                                                    IF Globals.enableDryCycle THEN
                                                        Globals.dryCycleCount := Globals.dryCycleCount + 1;     
                                                    ELSE
                                                        Globals.bagsMadeCount := Globals.bagsMadeCount + 1; 
                                                    END_IF
													IF enableBagOpen THEN
                                                        state := HEAD_STATES.OpenBag;
                                                    ELSE
                                                        state := HEAD_STATES.FinishCycle;
                                                    END_IF
                                                    
                                                            
                                                    
                                
    HEAD_STATES.OpenBag :                            // Close jaw to grab the bag
                                                    openBagSubState := BAG_OPEN_ASSIST_STATES.MoveJawIn;
                                                    state := HEAD_STATES.OpeningBag;
                                                    
                                                    
    HEAD_STATES.OpeningBag :                        // Open jaw and grab onto the bag
                                                    IF openBagSubState = BAG_OPEN_ASSIST_STATES.Done THEN
                                                        state := HEAD_STATES.OpenedBag;
                                                        openBagSubState := BAG_OPEN_ASSIST_STATES.Idle;
													ELSIF openBagSubState = BAG_OPEN_ASSIST_STATES.FeedNewBag THEN
														state := HEAD_STATES.SealAndSeparateBag;
														openBagSubState := BAG_OPEN_ASSIST_STATES.Idle;
                                                    END_IF
                                                    
    HEAD_STATES.OpenedBag :                            // Move fingers in and to bag holding and reset cycle
                                                    IF (motorizedSealFlatteners.state = SEAL_FLATTENER_STATES.Idle OR NOT motorizedSealFlatteners.enable) //OR bagFailedToOpen
														 AND pressureBar.state = PRESSURE_BAR_STATES.JawOpened THEN
														state := HEAD_STATES.FinishCycle;
                                                    END_IF
	HEAD_STATES.FinishCycle :			//
													finishCycleSubState := FINISH_CYCLE_STATES.Start;
													state := HEAD_STATES.FinishingCycle;
	HEAD_STATES.FinishingCycle : 		//
													IF finishCycleSubState = FINISH_CYCLE_STATES.Done THEN
														state := HEAD_STATES.FinishedCycle;
														finishCycleSubState := FINISH_CYCLE_STATES.Idle;
													END_IF
	HEAD_STATES.FinishedCycle :			//
											HMIData.bagsMade.Increment();
											HMIData.resettableBagsMade.Increment();
                                            state := HEAD_STATES.Idle;
											filler.BaggerCycledAndReady();
											cycleTime := (TIME_TO_REAL(cycleTimer.ET) / 1000); 
											cycleTimer.IN := FALSE;
											IF HMIData.averageCycleTime = 0 THEN
												HMIData.averageCycleTime := cycleTime;
											ELSE
												HMIData.averageCycleTime := (cycleTime + HMIData.averageCycleTime) / 2;
											END_IF
											HMIData.inCycle := FALSE;
											//bagFailedToOpen := FALSE;
											IF HMIData.factoryTestMode AND NOT HMIData.stopMachine THEN
												IF (HMIData.bagsMade.count >= 1000) THEN
													factoryTestModeKeepCycling := FALSE;
													HMIData.factoryTestMode := FALSE;
												ELSE
													factoryTestModeKeepCycling := TRUE;
												END_IF
											END_IF	
											
    HEAD_STATES.StartHoming :            // 
                                            passthrough.HomeEndStop();
                                            state := HEAD_STATES.Homing;                                        
    
    HEAD_STATES.Homing :                // 
                                            IF passthrough.state = PASSTHROUGH_SERVO_STATES.HomeComplete THEN
                                                state := HEAD_STATES.HomingComplete;       
                                            END_IF
                                            
    HEAD_STATES.HomingComplete :        // 
                                            homeJawPB := FALSE;
                                            state := HEAD_STATES.Idle;
											//HMIData.passthroughSetting := 6.0;
											setPassthroughPB := TRUE;
    
    HEAD_STATES.MovePassthrough :        // 
                                            pressureBar.AutoMovingPassthrough();
                                            passthrough.MovePassthrough(passthroughSetting);
                                            state := HEAD_STATES.MovingPassthrough;
    
    HEAD_STATES.MovingPassthrough :    IF passthrough.state = PASSTHROUGH_SERVO_STATES.PassthroughMovedIn OR passthrough.state = PASSTHROUGH_SERVO_STATES.PassthroughMovedOut THEN
                                                state := HEAD_STATES.MovedPassthrough;     
                                            END_IF
                                            
    HEAD_STATES.MovedPassthrough :        // 
                                            pressureBar.AutoDoneMovingPassthrough();
                                            state := HEAD_STATES.Idle;
											setPassthroughPB := FALSE;
                                                    
    HEAD_STATES.Fault :                     hmiLight.TurnOff();
											HMIData.inCycle := FALSE;
											cycleTimer.IN := FALSE;
											bagDelivery.bagFeedMasterMotor.SetRearMotorToEncoderFollowing();
											sealAndSeparateSubState := SEAL_SEPARATE_STATES.Idle;
											releaseAndFeedSubState := RELEASE_FEED_STATES.Idle;
											openBagSubState := BAG_OPEN_ASSIST_STATES.Idle;
											finishCycleSubState := FINISH_CYCLE_STATES.Idle;
											oVacOn := FALSE;
											filler.Reset();
											LPA.ManualOff();
											IBDRetractToDeflate.Reset();
											IBDRetractToEject.Reset();
											exitConveyorRun.Reset();
											externalExitConveyorRun.Reset();
											oRunPrinterRibbonUnwindMotor := FALSE;
											setPassthroughPB := FALSE;
											homeJawPB := FALSE;
											startCycle := FALSE;
											HMIData.initiateCycle := FALSE;
											factoryTestModeKeepCycling := FALSE;
											pressureBarCloseDelay.IN := FALSE;
											//bagOpened := FALSE;
                                                    
END_CASE

CASE sealAndSeparateSubState OF
    SEAL_SEPARATE_STATES.Idle : 
	
	SEAL_SEPARATE_STATES.BringInIBD : 				// Bring in IBD if enabled
													IF enableIBDDeflate THEN
														IBDRetractToDeflate.Trigger();
													END_IF 
													
													sealAndSeparateSubState := SEAL_SEPARATE_STATES.WaitForJawCloseDelay;
	
	SEAL_SEPARATE_STATES.WaitForJawCloseDelay : 	// Wait for jaw close delay. 
													IF pressureBar.enable THEN
														LPA.ManualOff();
														pressureBarCloseDelay.IN := TRUE;
														IF (pressureBarCloseDelay.Q OR HMIData.pressureBarCloseDelay = 0)
															AND (funnel.closed OR NOT funnel.enable)
															THEN
															sealAndSeparateSubState := SEAL_SEPARATE_STATES.MoveJawIn;
															pressureBarCloseDelay.IN := FALSE;
														END_IF
                                                    ELSE 
                                                        sealAndSeparateSubState := SEAL_SEPARATE_STATES.ReverseBag;
                                                    END_IF
        
    SEAL_SEPARATE_STATES.MoveJawIn :                // Perform actions as enabled - close jaw and move flatteners out. If jaw is disabled then go right to reverse bag
                                                    IF motorizedSealFlatteners.enable THEN
                                                        motorizedSealFlatteners.AutoMoveOut();
                                                    END_IF
                                                    
													pressureBar.AutoCloseJaw();
                                                    sealAndSeparateSubState := SEAL_SEPARATE_STATES.MovingJawIn;
                                                    
                                                    
                                                    
                                                    
                                                    
    SEAL_SEPARATE_STATES.MovingJawIn :                // If Jaw is in and flatteners out then move on
                                                    IF (motorizedSealFlatteners.state = SEAL_FLATTENER_STATES.MovedFlattenersOut OR NOT motorizedSealFlatteners.enable) 
                                                        AND (pressureBar.state = PRESSURE_BAR_STATES.JawClosed OR NOT pressureBar.enable)
                                                        THEN
                                                            sealAndSeparateSubState := SEAL_SEPARATE_STATES.MovedJawIn;    
                                                    END_IF
                                                                
    SEAL_SEPARATE_STATES.MovedJawIn :                // Will add sealing logic here
                                                    sealAndSeparateSubState := SEAL_SEPARATE_STATES.ReverseBag;
                                                    
    SEAL_SEPARATE_STATES.ReverseBag :                // Reverse bag if bag delivery enabled, otherwise open jaw
													IBDRetractToDeflate.Reset();
                                                    IF bagDelivery.enable THEN
                                                        bagDelivery.AutoReverseBag();
                                                        sealAndSeparateSubState := SEAL_SEPARATE_STATES.ReversingBag;
                                                    ELSE sealAndSeparateSubState := SEAL_SEPARATE_STATES.Done;    
                                                    END_IF
                                                                    
    SEAL_SEPARATE_STATES.ReversingBag :                // 
													IF NOT HMIData.separateBeforeSeal THEN
														sealTimer.PT := TO_TIME(HMIData.sealBarDwell * 1000);
														sealTimer.IN := TRUE;
														IF NOT sealTimer.Q THEN
															oSealBarExtend := TRUE;
															oSealBarRetract := FALSE;
														ELSE 
															
															oSealBarExtend := FALSE;
															oSealBarRetract := TRUE;
															
														END_IF
													END_IF

                                                    IF (motorizedSealFlatteners.state = SEAL_FLATTENER_STATES.MovedFlattenersOut OR NOT motorizedSealFlatteners.enable) 
                                                        AND (pressureBar.state = PRESSURE_BAR_STATES.JawClosed OR NOT pressureBar.enable)
                                                        AND (bagDelivery.state = BAG_DELIVERY_STATES.ReverseDone OR NOT bagDelivery.enable)
														AND (sealTimer.Q OR HMIData.separateBeforeSeal)
                                                        THEN
															IF NOT HMIData.separateBeforeSeal THEN
																HMIData.sealBarCycles.Increment();
															END_IF
															
															sealTimer.IN := FALSE;
                                                            sealAndSeparateSubState := SEAL_SEPARATE_STATES.Reversedbag;
                                                    END_IF
    SEAL_SEPARATE_STATES.Reversedbag :                // 
                                                    sealAndSeparateSubState := SEAL_SEPARATE_STATES.SealBag;
													
	SEAL_SEPARATE_STATES.SealBag:					
													IF HMIData.separateBeforeSeal THEN
														sealTimer.PT := TO_TIME(HMIData.sealBarDwell * 1000);
														sealTimer.IN := TRUE;
														IF NOT sealTimer.Q THEN
															oSealBarExtend := TRUE;
															oSealBarRetract := FALSE;
														ELSE 
															sealTimer.IN := FALSE;
															oSealBarExtend := FALSE;
															oSealBarRetract := TRUE;
															HMIData.sealBarCycles.Increment();
															sealAndSeparateSubState := SEAL_SEPARATE_STATES.Done;
														END_IF
													ELSE
														sealAndSeparateSubState := SEAL_SEPARATE_STATES.Done;
													END_IF
													
																				
                                                    
    SEAL_SEPARATE_STATES.Done :                        // 
                                                    
                                    
    SEAL_SEPARATE_STATES.Fault :
END_CASE


CASE releaseAndFeedSubState OF
    RELEASE_FEED_STATES.Idle :                        //
                                                        
    RELEASE_FEED_STATES.MoveJawOutAndDropBag :        // 
                                                    IF (motorizedSealFlatteners.state = SEAL_FLATTENER_STATES.MovedFlattenersOut OR NOT motorizedSealFlatteners.enable) 
                                                        AND (pressureBar.state = PRESSURE_BAR_STATES.JawClosed OR NOT pressureBar.enable)
                                                        AND ((bagDelivery.state = BAG_DELIVERY_STATES.ReverseDone) OR Globals.enableDryCycle)
                                                        OR (bagDelivery.state =  BAG_DELIVERY_STATES.WaitingForPrinter AND zebraPrinter.enable)
                                                        OR NOT bagDelivery.enable
                                                        THEN
                                                            IF motorizedSealFlatteners.enable THEN
                                                                motorizedSealFlatteners.AutoMoveToClearance();
                                                            END_IF
                                                            
                                                            IF pressureBar.enable THEN
                                                                pressureBar.AutoOpenJaw();
                                                            END_IF
                                                            
															IF enableBagOpen THEN
																bagOpenFingers.Release();
															END_IF
															
															IF enableIBDEject THEN
																IBDRetractToEject.Trigger();
															END_IF
															
															IF enableLoadPlate THEN
																rearLoadPlateRetract.Trigger();
															END_IF
															
															IF TO_DINT(HMIData.exitConveyorDwell) <> 0 THEN
																exitConveyorRun.Trigger();
															END_IF
															
															IF TO_DINT(HMIData.externalExitConveyorDwell) <> 0 THEN
																externalExitConveyorRun.Trigger();
															END_IF
															
															IF enableLabelSideUp THEN
																forwardLoadPlateRetract.Trigger();
																loadShelfExtend.Trigger();
															END_IF
															
															IF HMIData.lpaBagEjectAssistEnable THEN
																LPA.ManualOn();
															END_IF
                                                           bagDropTimer.IN := TRUE;
														   releaseAndFeedSubState := RELEASE_FEED_STATES.MovingJawOutAndDroppingBag;
                                                    END_IF
													
	 RELEASE_FEED_STATES.MovingJawOutAndDroppingBag :
														 // If printer is enabled then perform printer operation of bag delivery, otherwise just feed new bag out.
                                                            // In the case that bagDelivery is disabled then we're done with release and feed
                                                        IF bagDropTimer.Q 
															AND (motorizedSealFlatteners.state = SEAL_FLATTENER_STATES.MovedFlattenersToBagFeed OR NOT motorizedSealFlatteners.enable)
															THEN   
															bagDropTimer.IN := FALSE;
															IBDRetractToEject.Reset();
															IBDRetractToDeflate.Reset();
															IF bagDelivery.enable AND NOT zebraPrinter.enable THEN
                                                                bagDelivery.AutoFeedBagOut();
																LPA.ManualOff();
																IF HMIData.lpaDuringBagFeedEnable THEN
																	LPA.ManualOn();
																END_IF
                                                                releaseAndFeedSubState := RELEASE_FEED_STATES.MovingJawOutAndFeedingBag;
                                                            ELSIF bagDelivery.enable AND zebraPrinter.enable THEN
                                                                bagDelivery.AutoWaitForPrinter();
																LPA.ManualOff();
                                                                releaseAndFeedSubState := RELEASE_FEED_STATES.WaitForPrinter;
                                                            ELSE 
                                                                releaseAndFeedSubState := RELEASE_FEED_STATES.Done;
                                                            END_IF
                                                            (*{warning 'TODO: This is a hack to use HPA as LPA'}
														    HPA.DwellSetting := 500;		// Get rid on this - ha
													        HPA.Trigger();*)												
    													END_IF
														
    RELEASE_FEED_STATES.WaitForPrinter :            // Data Ready means the printer has a label and we're all set to print
                                                    IF zebraPrinter.state = PRINTER_STATES.DataReady THEN
                                                        releaseAndFeedSubState := RELEASE_FEED_STATES.FeedToOffset;
                                                    END_IF
                                                    
    RELEASE_FEED_STATES.FeedToOffset :                // This starts feeding to the print offset
													IF (motorizedSealFlatteners.state = SEAL_FLATTENER_STATES.MovedFlattenersToBagFeed OR NOT motorizedSealFlatteners.enable) THEN
														bagDelivery.AutoPrinterReady();
                                                    	releaseAndFeedSubState := RELEASE_FEED_STATES.FeedingToOffset;
													END_IF
                                                    
                                                        
    RELEASE_FEED_STATES.FeedingToOffset :            // Once offset done start printing
                                                    IF bagDelivery.state = BAG_DELIVERY_STATES.FedToPrintOffset THEN
                                                        releaseAndFeedSubState := RELEASE_FEED_STATES.StartPrinting;
                                                    END_IF                                            
    
    RELEASE_FEED_STATES.StartPrinting :                // Printer starts print cycle and bag delivery starts moving at print speed
                                                    
                                                    //bagDelivery.AutoStartPrintFeed();
													zebraPrinter.AutoPrintNow();
                                                    
                                                    releaseAndFeedSubState := RELEASE_FEED_STATES.SendPrintSignal;                                            

    RELEASE_FEED_STATES.SendPrintSignal:            // 
                                                    //IF bagDelivery.state =     BAG_DELIVERY_STATES.FeedingAtPrintSpeed THEN
													//zebraPrinter.AutoSendPrintSignal();
													IF zebraPrinter.printHeadDebounced THEN
														bagDelivery.AutoStartPrintFeed();
														zebraPrinter.AutoSendPrintSignal();
														barcodeVerifier.Trigger();
                                                        //bagDelivery.AutoStartPrintFeed();
														//bagDelivery.AutoStartPrintFeed();
                                                        //zebraPrinter.AutoSendPrintSignal();
														
                                                        releaseAndFeedSubState := RELEASE_FEED_STATES.Printing;
                                                    END_IF                                        

    RELEASE_FEED_STATES.Printing :                // 
													
                                                    IF zebraPrinter.state = PRINTER_STATES.DonePrinting THEN
                                                        releaseAndFeedSubState := RELEASE_FEED_STATES.StopPrinting;
                                                    END_IF
                                                    
    RELEASE_FEED_STATES.StopPrinting :                // Tell bag delivery it's okay to feed out the rest of the bag and the printer that it can prep itself for the next print
                                                    bagDelivery.AutoPrinterDone();
                                                    zebraPrinter.AutoAckPrintDone();
													IF HMIData.lpaDuringBagFeedEnable THEN
														LPA.ManualOn();
													END_IF
													
                                                    releaseAndFeedSubState := RELEASE_FEED_STATES.MovingJawOutAndFeedingBag;
                                                                                
                                                                                                            
    RELEASE_FEED_STATES.MovingJawOutAndFeedingBag :    // 
    
													
													IF (bagdelivery.state = BAG_DELIVERY_STATES.Ready OR NOT bagdelivery.enable)
                                                        AND (motorizedSealFlatteners.state = SEAL_FLATTENER_STATES.MovedFlattenersToBagFeed OR NOT motorizedSealFlatteners.enable) 
                                                        AND (pressureBar.state = PRESSURE_BAR_STATES.JawOpened OR NOT pressureBar.enable)
                                                        THEN
															IF LPA.DwellSetting = 0 THEN
																LPA.ManualOff();
															END_IF
															IBDRetractToEject.Reset();
                                                            releaseAndFeedSubState := RELEASE_FEED_STATES.MovedJawOutAndFedBag;
                                                    END_IF
                                                    
    RELEASE_FEED_STATES.MovedJawOutAndFedBag :      // Wait until bag is fed out before triggering barcode fail.
													IF barcodeVerifier.barcodeFault THEN
														barcodeVerificationFailed.Trigger();
													END_IF 
													releaseAndFeedSubState := RELEASE_FEED_STATES.Done;
    RELEASE_FEED_STATES.Done :
    RELEASE_FEED_STATES.Fault :
END_CASE

CASE openBagSubState OF
    BAG_OPEN_ASSIST_STATES.Idle :                    // 
                                                    
                                                    
                                                    
    BAG_OPEN_ASSIST_STATES.MoveJawIn :                // Close jaw against bag. In the future we may also start vacuum here
                                                    pressureBar.AutoCloseJaw();
													(*HPA.DwellSetting := 80;
													HPA.Trigger();*)
													IF HPA.DwellSetting <> 0 THEN
														HPA.Trigger();	
													END_IF
													
													//oVacOn := TRUE; // Hard coded for now, this is vacuum
                                                    openBagSubState := BAG_OPEN_ASSIST_STATES.MovingJawIn;        
                                                    
                                                    
    BAG_OPEN_ASSIST_STATES.MovingJawIn :            // Move on once jaw is closed
                                                    IF (pressureBar.state = PRESSURE_BAR_STATES.JawClosed) OR NOT pressureBar.enable THEN
                                                        openBagSubState := BAG_OPEN_ASSIST_STATES.MovedJawIn;        
                                                    END_IF
                                                    
                                                    
    BAG_OPEN_ASSIST_STATES.MovedJawIn :                // Hold onto the bag with vacuum to build suction
                                                    vacuumHoldTimer.IN := TRUE;
													oVacOn := TRUE; // Hard coded for now, this is vacuum
													IF vacuumHoldTimer.Q THEN
														openBagSubState := BAG_OPEN_ASSIST_STATES.MoveJawOut; 
														vacuumHoldTimer.IN := FALSE;
													END_IF
                                                                   
                                                    
                                                    
    BAG_OPEN_ASSIST_STATES.MoveJawOut :                // Open the jaw and move seal flatteners in and to bag holding
                                                    pressureBar.AutoOpenJaw();
													motorizedSealFlatteners.AutoMoveIn();
                                                    openBagSubState := BAG_OPEN_ASSIST_STATES.MovingJawOutAndGrab;
                                                    
                                                    
    BAG_OPEN_ASSIST_STATES.MovingJawOutAndGrab :    // Once everything that is enabled is homed finish cycle 
													bagOpenFingerDelay.IN := TRUE;
													IF bagOpenFingerDelay.Q THEN
														bagOpenFingers.Grab();
														bagOpenFingerDelay.IN := FALSE;

														openBagSubState := BAG_OPEN_ASSIST_STATES.CheckForSuccessfulBagGrab;
													END_IF
													  

	BAG_OPEN_ASSIST_STATES.CheckForSuccessfulBagGrab : 	//
														IF bagOpenRetryCount < bagOpenRetrySetting THEN
															bagOpenCheckDelay.IN := TRUE;
															IF bagOpenCheckDelay.Q THEN
																IF bagOpenFingers.CheckIfBagGrabbed(TRUE) THEN // This method checks to see if the bag is grabbed and returns true if so.
																	openBagSubState := BAG_OPEN_ASSIST_STATES.BagOpened;
																	motorizedSealFlatteners.AutoMoveIn();
																ELSE 
																	openBagSubState := BAG_OPEN_ASSIST_STATES.BagFailedToOpen;
																END_IF
																bagOpenCheckDelay.IN := FALSE;
															END_IF
														ELSE 
															motorizedSealFlatteners.AutoMoveToBagHolding();
															openBagSubState := BAG_OPEN_ASSIST_STATES.MovingJawOutAfterGrab;
														END_IF
													  
	BAG_OPEN_ASSIST_STATES.BagFailedToOpen :			// 
														bagOpenFingers.Release();
														bagOpenRetryCount := bagOpenRetryCount + 1;
														IF bagOpenRetryCount < bagOpenRetrySetting THEN
															openBagSubState := BAG_OPEN_ASSIST_STATES.MoveJawIn;
														ELSIF HMIData.bagOpenFeedNewBagCount < HMIData.bagOpenFeedNewBagSetting THEN
															HMIData.bagOpenFeedNewBagCount := HMIData.bagOpenFeedNewBagCount + 1;
															bagOpenRetryCount := 0;
															motorizedSealFlatteners.AutoMoveOut();
															oVacOn := FALSE;
															openBagSubState := BAG_OPEN_ASSIST_STATES.FeedNewBag;
															
														ELSE 
															//IF (motorizedSealFlatteners.state = SEAL_FLATTENER_STATES.Idle OR NOT motorizedSealFlatteners.enable) THEN
																motorizedSealFlatteners.AutoMoveToBagHolding();
																bagFailedToOpen.Trigger();
																
																openBagSubState := BAG_OPEN_ASSIST_STATES.MovingJawOutAfterGrab;
																bagOpenRetryCount := 0; 
																HMIData.bagOpenFeedNewBagCount := 0;
																HMIData.bagsRejectedTotal.Increment();
																Globals.rejectedBagCount := Globals.rejectedBagCount + 1;
															//END_IF
															
														END_IF
	
	BAG_OPEN_ASSIST_STATES.BagOpened :					//
														bagOpened := TRUE;
                                                    	motorizedSealFlatteners.AutoMoveToBagHolding();
														bagOpenRetryCount := 0;
														HMIData.bagOpenFeedNewBagCount := 0;
														
														openBagSubState := BAG_OPEN_ASSIST_STATES.MovingJawOutAfterGrab; 
														
                                      
    BAG_OPEN_ASSIST_STATES.MovingJawOutAfterGrab :		// 
														IF (pressureBar.state = PRESSURE_BAR_STATES.JawOpened OR NOT pressureBar.enable) 
															AND (motorizedSealFlatteners.state = SEAL_FLATTENER_STATES.Idle OR NOT motorizedSealFlatteners.enable)
															THEN
																openBagSubState := BAG_OPEN_ASSIST_STATES.MovedJawOut;        
														END_IF	 
														
	
	BAG_OPEN_ASSIST_STATES.MovedJawOut :            // 
														oVacOn := FALSE; 		// Hard coded for now, this is vacuum
														
														
														openBagSubState := BAG_OPEN_ASSIST_STATES.Done;

                                                             
                                                
	BAG_OPEN_ASSIST_STATES.FeedNewBag :   			//
													IF (motorizedSealFlatteners.state = SEAL_FLATTENER_STATES.Idle OR NOT motorizedSealFlatteners.enable) THEN
														state := HEAD_STATES.SealAndSeparateBag;
													END_IF
													
													
                                                
    BAG_OPEN_ASSIST_STATES.Done :                    // 
                                                            
    BAG_OPEN_ASSIST_STATES.Fault :                    //
													

END_CASE

CASE finishCycleSubState OF
	FINISH_CYCLE_STATES.Idle:								//
	
	FINISH_CYCLE_STATES.Start :								//
															IF funnel.enable THEN
																finishCycleSubState := FINISH_CYCLE_STATES.OpenFunnel;
															ELSIF enableBagOpen THEN
																finishCycleSubState := FINISH_CYCLE_STATES.Done;
															ELSE
																IF motorizedSealFlatteners.enable THEN
																	finishCycleSubState := FINISH_CYCLE_STATES.BringSealFlattenersInAndDown;
																ELSE
																	finishCycleSubState := FINISH_CYCLE_STATES.Done;
																END_IF
															END_IF
															IF LPA.DwellSetting <> 0 THEN
																LPA.Trigger();
															END_IF
	
	FINISH_CYCLE_STATES.OpenFunnel :						//
															IF LPA.DwellSetting <> 0 THEN
																LPA.Trigger();
															END_IF
															funnel.OpenNow();
															finishCycleSubState := FINISH_CYCLE_STATES.OpeningFunnel;
	
	FINISH_CYCLE_STATES.OpeningFunnel :						//
															IF funnel.opened THEN
																finishCycleSubState := FINISH_CYCLE_STATES.OpenedFunnel;
															END_IF
	
	FINISH_CYCLE_STATES.OpenedFunnel :						//
															//IF enableBagOpen THEN
																IF iLefttFingerBagPresent AND iRightFingerBagPresent THEN
																	finishCycleSubState := FINISH_CYCLE_STATES.Done;
																ELSE
																	IF bagOpenRetryCount < bagOpenRetrySetting THEN
																		bagOpenRetryCount := bagOpenRetryCount + 1;
																		funnel.CloseNow();
																		finishCycleSubState := FINISH_CYCLE_STATES.ClosingFunnelForRetry;
																	ELSE
																		bagFailedToOpen.Trigger();
																		funnel.CloseNow();
																		bagOpenRetryCount := 0; 
																		HMIData.bagsRejectedTotal.Increment();
																		finishCycleSubState := FINISH_CYCLE_STATES.Done;
																	END_IF
																END_IF
															ELSE
																IF motorizedSealFlatteners.enable THEN
																	finishCycleSubState := FINISH_CYCLE_STATES.BringSealFlattenersToBagHolding;
																ELSE
																	finishCycleSubState := FINISH_CYCLE_STATES.Done;
																END_IF
															//END_IF
	
	FINISH_CYCLE_STATES.ClosingFunnelForRetry :				//
															IF funnel.closed THEN
																finishCycleSubState := FINISH_CYCLE_STATES.Start;
															END_IF												
	
	FINISH_CYCLE_STATES.BringSealFlattenersInAndDown :		//
															motorizedSealFlatteners.AutoMoveToHandLoad();
															finishCycleSubState := FINISH_CYCLE_STATES.BringingSealFlattenersInAndDown;
	
	FINISH_CYCLE_STATES.BringingSealFlattenersInAndDown :	//
															IF motorizedSealFlatteners.state = SEAL_FLATTENER_STATES.Idle THEN
																finishCycleSubState := FINISH_CYCLE_STATES.SealFlattenersInAndDown;
															END_IF
	
	FINISH_CYCLE_STATES.SealFlattenersInAndDown :			//
															finishCycleSubState := FINISH_CYCLE_STATES.Done;
	
	FINISH_CYCLE_STATES.BringSealFlattenersToBagHolding:	//
															motorizedSealFlatteners.AutoMoveToBagHolding();
															finishCycleSubState := FINISH_CYCLE_STATES.BringingSealFlattenersToBagHolding;
	
	FINISH_CYCLE_STATES.BringingSealFlattenersToBagHolding: //
															IF motorizedSealFlatteners.state = SEAL_FLATTENER_STATES.Idle THEN
																finishCycleSubState := FINISH_CYCLE_STATES.SealFlattenersAtBagHolding;
															END_IF
																
	FINISH_CYCLE_STATES.SealFlattenersAtBagHolding : 		//
															finishCycleSubState := FINISH_CYCLE_STATES.Done;
	
	FINISH_CYCLE_STATES.Done :								//
															bagOpenRetryCount := 0;
														
	
	FINISH_CYCLE_STATES.Fault :
	
	
END_CASE
HMIData.initiateCycle := FALSE;

END_FUNCTION_BLOCK

// FBs/Components/BaseComponentFB
FUNCTION_BLOCK BaseComponentFB IMPLEMENTS IComponentStatus
VAR_INPUT
	enable : BOOL;                    // Enable
END_VAR
VAR_OUTPUT
END_VAR
VAR
	_mode : DEVICE_MODES;            // Auto-SemiAuto-Manual
    _ready : BOOL;                    // Ready to be controlled
	_reset : BOOL;
	enableONS : R_TRIG;
	resetONS : R_TRIG;
	autoModeSelected : BOOL;
    semiAutoModeSelected : BOOL;
    manualModeSelected : BOOL;
END_VAR

//	Function Block: BaseComponentFB
//	Description:  Extend this FB for each component as it contains the basic variables and logic that all components must share
//	In all extended FBs you must run the parent logic with SUPER^()
//	Created by: Ben Hess
//	Created Date: Friday, June 1, 2018


enableONS(CLK := enable);
resetONS(CLK := _reset);

autoModeSelected := (_mode = DEVICE_MODES.Auto);
semiAutoModeSelected := (_mode = DEVICE_MODES.SemiAuto);
manualModeSelected := (_mode = DEVICE_MODES.Manual);
IF _reset THEN
	_reset := FALSE;
END_IF

PROPERTY Ready : BOOL
GET
Ready := _ready;
END_GET
SET
_ready := Ready;
END_SET
END_PROPERTY

METHOD Reset : BOOL
VAR_INPUT
END_VAR
_reset := TRUE;
END_METHOD

PROPERTY Mode : DEVICE_MODES
GET
Mode := _mode;
END_GET
SET
_mode := Mode;
END_SET
END_PROPERTY

END_FUNCTION_BLOCK

// Pro18_1174/Application/Interfaces/IComponentStatus
INTERFACE IComponentStatus

PROPERTY Mode : DEVICE_MODES
SET
END_SET
GET
END_GET
END_PROPERTY

PROPERTY Ready : BOOL
GET
END_GET
SET
END_SET
END_PROPERTY

END_INTERFACE

// ElectricMachine/Application/Interfaces/IComponentStatus
INTERFACE IComponentStatus

PROPERTY Mode : DEVICE_MODES
GET
END_GET
SET
END_SET
END_PROPERTY

PROPERTY Ready : BOOL
SET
END_SET
GET
END_GET
END_PROPERTY

END_INTERFACE

// FBs/Components/MotorizedSealFlattenersFB_BagFeed
FUNCTION_BLOCK MotorizedSealFlattenersFB_BagFeed EXTENDS BaseComponentFB IMPLEMENTS IComponentStatus
VAR_INPUT
    {warning 'TODO: Make a struct for some of these - too many inputs'}
	sealFlattenersVerticalAxis : ICylinder();
    clearanceOffset : REAL := 2.0;        // Clearance Offset in inches
	bagFeedPosition : REAL;
    inSetpoint : REAL := 1.25;            // In setpoint in inches
    outSetpoint : REAL := 17.7;            // Out (sealing) setpoint in inches
    bagHoldingSetpoint : REAL := 17;    // Bag holding setpoint in inches            
    clearanceSpeed : INT := 3000;        // Speed to move in clearance move
    moveInSpeed : INT := 3000;            // Speed to move in in move
    moveOutSpeed : INT := 1000;            // Speed to move in out move
    moveBagHoldingSpeed : INT := 1000;    // Speed to move in bag holding move
    fingersUpSetpoint : REAL := 0;     // Fingers Up setpoint in inches
    fingersDownSetpoint : REAL := 1.1; // Fingers down setpoint in inches
    moveFingersSpeed : INT := 2000;        // Speed to move fingers
    horizontalAxisAccel : INT := 1000;    // Accel setpoint for horizontal axis
    horizontalAxisDecel : INT := 1000;    // Decel Setpoint for horizontal axis
    verticalAxisAccel : INT := 150;    // Accel setpoint for vertical axis
    verticalAxisDecel : INT := 150;    // Decel Setpoint for vertical axis
    testMovePB : BOOL;
    testMoveSP : REAL;
    stopPB : BOOL;
    startPB : BOOL;
    nextSeqPB : BOOL;
    delay : TON := (PT:= T#300MS);
	fingersDownDelay : Standard.TON := (PT := T#200MS);
	sealFlattenerMotorCommFailInput : BOOL;
	manualPosSetpoint : REAL;
	
END_VAR
VAR_IN_OUT
	jogIn : BOOL;
	jogOut : BOOL;
	raiseService : BOOL;
	lowerService : BOOL;
	moveToManualSetpoint : BOOL;
END_VAR
VAR_OUTPUT
    state : SEAL_FLATTENER_STATES;
END_VAR
VAR
    //pressureBarMotor : FB_FestoMotor();
    //sealFlattenersVerticalAxisMotor : FB_AppliedMotionStepServoRTU();
	jogInONS: FB_ONS;
	jogOutONS: FB_ONS;
	jogSpeed : INT := 100;
    sealFlattenersHorizontalAxisMotor : FB_AppliedMotionStepServoEIPBaseQX();
	defaultCurrentMSF : DINT := 150;
	outCurrentMSF : DINT := 150;
	bagHoldingCurrentMSF : DINT := 85;
    enableMotorizedSealFlattenersONS : R_TRIG();
	bagDropDelay : Standard.TON := (PT := T#1S);    
    _amMoveOut : BOOL;                // Auto mode move out command
	_amMoveIn : BOOL;
    _amMoveClearance : BOOL;            // Auto mode move Clearance command
    _amMoveInToBagHolding : BOOL;    // Auto mode move in then bag holding command
	_amMoveHandLoad : BOOL;			// Auto move to hand load positon command
	handLoadRequested : BOOL;
END_VAR

//    Function Block:  MotorizedSealFlattenersFB
//    Description: State machine and motor management for motorized seal flateners
//    Currently, this code requires one to use the Oriental drive with pre-programmed 
//    sequence for the horizontal axis
//    Created by: Ben Hess
//    Created Date: Friday, April 6, 2018
SUPER^();
// Setup and execute 2 motor axis'

// Temporary delay between states for testing
fingersDownDelay();
bagDropDelay(PT := TO_TIME(HMIData.bagDropTime * 1000));
delay();
jogInONS(CLK := jogIn);
jogOutONS(CLK := jogOut);
IF autoModeSelected THEN
    delay.PT := T#300MS;
ELSE
    delay.PT := T#750MS;
END_IF

outSetpoint := HMIData.bagWidth + 0.2;
bagHoldingSetpoint := HMIData.bagWidth;

// Setup the vertical axis motor
sealFlattenersVerticalAxis.Execute();

// Setup the horizontal axis motor 
(*
sealFlattenersHorizontalAxisMotor(modbusInBuffer := OrientalMotorModbusRead,
                stepsPerInchSetpoint := 125,
                reversePolarity := FALSE,
                operatingCurrentDefault := 500,
                modbusCommandOutBuffer := OrientalMotorCommandWrites,
                modbusParametersOutBuffer := OrientalMotorParameterWrites,
                triggerCommandWrite => OrientalMotorTriggerCommandWrite,
                triggerParameterWrite => OrientalMotorTriggerParameterWrite);                
sealFlattenersHorizontalAxisMotor.Execute();
*)

sealFlattenersHorizontalAxisMotor(ptrEIPInputs := ADR(sealFlattenerHorizontalMotorInputs),
                ptrEIPOutputs := ADR(sealFlattenerHorizontalMotorOutputs),
                stepsPerInchSetpoint := Globals.STEPS_PER_INCH_SEAL_FLATTENER_HORIZONTAL_AXIS_MOTOR,
                faultHandler := PRG_Bagger.faultHandler,
				reversePolarity := TRUE, 
				defaultCurrentSetpoint := defaultCurrentMSF, 
				commFail := sealFlattenerMotorCommFailInput,
				isHomable := TRUE);
				
sealFlattenersHorizontalAxisMotor.Execute();

//Report as ready if mode is auto and we're not faulted
_ready := (_mode = DEVICE_MODES.Auto) AND NOT (state = SEAL_FLATTENER_STATES.Fault);

enableMotorizedSealFlattenersONS(CLK := enable);
IF stopPB THEN
    sealFlattenersHorizontalAxisMotor.Stop();
    stopPB := FALSE;
END_IF

IF startPB AND semiAutoModeSelected THEN 
    //sealFlattenersHorizontalAxisMotor.StartOperation();
    startPB := FALSE;
END_IF

IF nextSeqPB THEN 
    //sealFlattenersHorizontalAxisMotor.NextSequence();
    nextSeqPB := FALSE;
END_IF

IF testMovePB THEN
    sealFlattenersHorizontalAxisMotor.MoveToPosition(position := (testMoveSP), acceleration := 100, deceleration := 100, velocity := 600);
    testMovePB := FALSE;
END_IF

IF enableONS.Q OR resetONS.Q THEN 
    state := SEAL_FLATTENER_STATES.Idle;
	sealFlattenersHorizontalAxisMotor.Reset();
	_reset := FALSE;
	bagDropDelay.IN := FALSE;
	ClearCommands();
	handLoadRequested := FALSE;
END_IF

IF NOT enable THEN
    state := SEAL_FLATTENER_STATES.Fault;
END_IF

// State amchine for motorized seal flatteners
CASE state OF
    

    SEAL_FLATTENER_STATES.Idle :                                    //If enabled move to out
                                                                    IF enable AND semiAutoModeSelected OR (autoModeSelected AND _amMoveOut) THEN
                                                                        state := SEAL_FLATTENER_STATES.MoveFlattenersOut;
                                                                        ClearCommands();
                                                                    END_IF
																	
																	IF enable AND autoModeSelected AND _amMoveIn OR _amMoveInToBagHolding THEN
																	//IF enable AND autoModeSelected AND _amMoveIn THEN
																		sealFlattenersVerticalAxis.Retract();
																		state := SEAL_FLATTENER_STATES.MoveFlattenersIn;
																		ClearCommands();
																	END_IF
																	
																	IF jogInONS.OSR THEN
																		sealFlattenersHorizontalAxisMotor.MoveDistance(distance := -18, 
																									acceleration := horizontalAxisAccel, 
																									deceleration := horizontalAxisDecel, 
																									velocity := jogSpeed);
																	ELSIF jogOutONS.OSR THEN
																		sealFlattenersHorizontalAxisMotor.MoveDistance(distance := 18, 
																									acceleration := horizontalAxisAccel, 
																									deceleration := horizontalAxisDecel, 
																									velocity := jogSpeed);
																	ELSIF jogInONS.OSF OR jogOutONS.OSF THEN
																		sealFlattenersHorizontalAxisMotor.Stop();
																	END_IF
																	
																	IF raiseService THEN
																		sealFlattenersVerticalAxis.Retract();  
																		
																		raiseService := FALSE;
																	ELSIF lowerService THEN
																		sealFlattenersVerticalAxis.Extend();  
																		lowerService := FALSE;
																	END_IF
																	
																	IF moveToManualSetpoint THEN
																		sealFlattenersHorizontalAxisMotor.MoveToPosition(position := manualPosSetpoint, 
																									acceleration := horizontalAxisAccel, 
																									deceleration := horizontalAxisDecel, 
																									velocity := moveFingersSpeed);
																		moveToManualSetpoint := FALSE;
																	END_IF
																	
																	bagDropDelay.IN := FALSE;
																	
                                                                    
    SEAL_FLATTENER_STATES.MoveFlattenersOut :                        // Move flatteners to out position
                                                                
                                                                    //sealFlattenersHorizontalAxisMotor.StartOperation();
                                                                    sealFlattenersHorizontalAxisMotor.MoveToPositionTorque(position := outSetpoint, 
                                                                                                                        acceleration := horizontalAxisAccel,
                                                                                                                        deceleration := horizontalAxisDecel,
                                                                                                                        velocity := moveOutSpeed,
																														current := outCurrentMSF);                                                    
                                                                    state := SEAL_FLATTENER_STATES.MovingFlattenersOut;
                                                                    
                                                                    
    SEAL_FLATTENER_STATES.MovingFlattenersOut :                        // 
                                                                    delay.IN := TRUE;
                                                                    IF delay.Q THEN
																		IF sealFlattenersHorizontalAxisMotor.CommandAcknowledged AND sealFlattenersHorizontalAxisMotor.CurrentPosition >= (bagHoldingSetpoint - 1.5) THEN
																			state := SEAL_FLATTENER_STATES.MovedFlattenersOut;
                                                                        	delay.IN := FALSE; 
																		END_IF
                                                                    END_IF
                                                                    
    SEAL_FLATTENER_STATES.MovedFlattenersOut :                        // Move flatteners to clearance position state
                                                                    IF enable AND semiAutoModeSelected OR (autoModeSelected AND _amMoveClearance) THEN
                                                                        state := SEAL_FLATTENER_STATES.MoveFlattenersUpAndToClearance;
                                                                        ClearCommands();
                                                                    END_IF
    
    
    SEAL_FLATTENER_STATES.MoveFlattenersUpAndToClearance :                // Move flatteners to clearance position
                                                                    
                                                                    //sealFlattenersHorizontalAxisMotor.NextSequence();
                                                                    sealFlattenersHorizontalAxisMotor.MoveToPosition(position := (outSetpoint - clearanceOffset), 
                                                                                                                        acceleration := horizontalAxisAccel,
                                                                                                                        deceleration := horizontalAxisDecel,
                                                                                                                        velocity := moveOutSpeed);    
                                                                   	sealFlattenersVerticalAxis.Retract();                                                       
                                                                    state := SEAL_FLATTENER_STATES.MovingFlattenersUpAndToClearance;    
    
    
    
    SEAL_FLATTENER_STATES.MovingFlattenersUpAndToClearance :        delay.IN := TRUE;
                                                                    IF delay.Q THEN
																		IF sealFlattenersHorizontalAxisMotor.CommandAcknowledged AND sealFlattenersHorizontalAxisMotor.InPosition THEN
																			state := SEAL_FLATTENER_STATES.MovedFlattenersUpAndToClearance;    
                                                                        	delay.IN := FALSE;
																		END_IF
                                                                        
                                                                    END_IF
                                                                    
                                                                    
    SEAL_FLATTENER_STATES.MovedFlattenersUpAndToClearance :                // Move flatteners to up state
																	bagDropDelay.IN := TRUE;
																	IF bagDropDelay.Q THEN
																		state := SEAL_FLATTENER_STATES.MoveFlattenersToBagFeed;
																		bagDropDelay.IN := FALSE;
																	END_IF
                                                                    
                                                                    
																	
	SEAL_FLATTENER_STATES.MoveFlattenersToBagFeed :      			// Move flatteners to out of the way of the bag for feeding
																	IF (HMIData.baggerModelSelection = ModelSelection.Pro18) OR (HMIData.baggerModelSelection = ModelSelection.Pro18_02) THEN
																		IF (outSetpoint + clearanceOffset) <= 17.8 THEN
																			bagFeedPosition := (outSetpoint + clearanceOffset);
																		ELSE
																			bagFeedPosition := 17.8;
																		END_IF
																	ELSE
																		IF (outSetpoint + clearanceOffset) <= 23.8 THEN
																			bagFeedPosition := (outSetpoint + clearanceOffset);
																		ELSE
																			bagFeedPosition := 23.8;
																		END_IF
																	END_IF
																		
                                                                    sealFlattenersHorizontalAxisMotor.MoveToPosition(position := bagFeedPosition, 
                                                                                                                        acceleration := horizontalAxisAccel,
                                                                                                                        deceleration := horizontalAxisDecel,
                                                                                                                        velocity := moveInSpeed);              
                                                                    state := SEAL_FLATTENER_STATES.MovingFlattenersToBagFeed;
	
   SEAL_FLATTENER_STATES.MovingFlattenersToBagFeed :        			delay.IN := TRUE;
                                                                    IF delay.Q THEN
																		IF sealFlattenersHorizontalAxisMotor.CommandAcknowledged AND sealFlattenersHorizontalAxisMotor.InPosition THEN
																			state := SEAL_FLATTENER_STATES.MovedFlattenersToBagFeed;    
                                                                        	delay.IN := FALSE;
																		END_IF
                                                                    END_IF
																
	SEAL_FLATTENER_STATES.MovedFlattenersToBagFeed:					       // Move flatteners to up state
                                                                    IF enable AND semiAutoModeSelected OR (autoModeSelected AND (_amMoveInToBagHolding OR _amMoveIn OR _amMoveHandLoad)) THEN
                                                                        state := SEAL_FLATTENER_STATES.MoveFlattenersIn;
                                                                        //ClearCommands();
                                                                    END_IF
      

                               
                                                                    
    SEAL_FLATTENER_STATES.MoveFlattenersIn :                        // Move flatteners up and in
                                                                    //sealFlattenersHorizontalAxisMotor.NextSequence();    
                                                                    sealFlattenersHorizontalAxisMotor.MoveToPosition(position := inSetpoint, 
                                                                                                                        acceleration := horizontalAxisAccel,
                                                                                                                        deceleration := horizontalAxisDecel,
                                                                                                                        velocity := moveInSpeed);                                                    
                                                                    state := SEAL_FLATTENER_STATES.MovingFlattenersIn;
                                                                    
                                                                    
    SEAL_FLATTENER_STATES.MovingFlattenersIn :                        // If we did that command well move on 
                                                                        delay.IN := TRUE;
                                                                        IF delay.Q THEN
																			IF sealFlattenersHorizontalAxisMotor.CommandAcknowledged AND sealFlattenersHorizontalAxisMotor.InPosition THEN
																				state := SEAL_FLATTENER_STATES.MovedFlattenersIn;
                                                                           		delay.IN := FALSE;    
																			END_IF
                                                                        END_IF 
                                                                    
    SEAL_FLATTENER_STATES.MovedFlattenersIn :                        // Now that we're up and in move to down and 4 corners/bag holding
                                                                    IF enable AND semiAutoModeSelected OR (autoModeSelected AND (_amMoveInToBagHolding OR _amMoveHandLoad)) THEN
                                                                        state := SEAL_FLATTENER_STATES.MoveFlattenersDown;
																		IF _amMoveHandLoad THEN
																			 handLoadRequested := TRUE;
																		END_IF
                                                                        ClearCommands();
                                                                    END_IF    
																	
																	IF enable AND (autoModeSelected AND _amMoveOut) THEN
																		sealFlattenersHorizontalAxisMotor.MoveToPosition(position := outSetpoint, 
                                                                                                                        acceleration := horizontalAxisAccel,
                                                                                                                        deceleration := horizontalAxisDecel,
                                                                                                                        velocity := moveInSpeed);                                                    
                                                                    	state := SEAL_FLATTENER_STATES.Idle;
																		ClearCommands();
																	END_IF
    
    SEAL_FLATTENER_STATES.MoveFlattenersDown :            // Do moves for down and bag holding
                                                                        
                                                                        sealFlattenersVerticalAxis.Extend();
                                                                                                                                                                                
                                                                        state := SEAL_FLATTENER_STATES.MovingFlattenersDown;
                                                                        
    SEAL_FLATTENER_STATES.MovingFlattenersDown :            
                                                                        //IF sealFlattenersVerticalAxis.CommandAcknowledged AND sealFlattenersVerticalAxis.InPosition THEN
                                                                       	fingersDownDelay.IN := TRUE;
																	  	IF fingersDownDelay.Q THEN
																			state := SEAL_FLATTENER_STATES.MovedFlattenersDown;
																			fingersDownDelay.IN := FALSE;
																		END_IF 
																		
                                                                        //END_IF 
                                                                        
	SEAL_FLATTENER_STATES.MovedFlattenersDown :            			IF handLoadRequested THEN
																		state := SEAL_FLATTENER_STATES.Idle;
																		handLoadRequested := FALSE;
																	ELSE
																		state := SEAL_FLATTENER_STATES.MoveFlattenersToBagHolding;
																	END_IF
																	
                                                                    
                                                                    
    SEAL_FLATTENER_STATES.MoveFlattenersToBagHolding :            // Do moves for down and bag holding
                                                                        //sealFlattenersHorizontalAxisMotor.NextSequence();    
                                                                        sealFlattenersHorizontalAxisMotor.MoveToPositionTorque(position := bagHoldingSetpoint, 
                                                                                                                        acceleration := horizontalAxisAccel,
                                                                                                                        deceleration := horizontalAxisDecel,
                                                                                                                        velocity := moveBagHoldingSpeed,
																														current := bagHoldingCurrentMSF);                                                
                                                                        state := SEAL_FLATTENER_STATES.MovingFlattenersToBagHolding;
                                                                        
    SEAL_FLATTENER_STATES.MovingFlattenersToBagHolding :            delay.IN := TRUE;
                                                                        IF delay.Q THEN
																			IF sealFlattenersHorizontalAxisMotor.CommandAcknowledged THEN
																				state := SEAL_FLATTENER_STATES.MovedFlattenersToBagHolding;
                                                                            	delay.IN := FALSE; 
																			END_IF   
                                                                        END_IF 
                                                                        
    SEAL_FLATTENER_STATES.MovedFlattenersToBagHolding :            state := SEAL_FLATTENER_STATES.Idle;
																		HMIData.motorizedSealFlattenerCycles.Increment();
                                                                        Globals.motorizedSealFlattenersCount := Globals.motorizedSealFlattenersCount +1;
                                                                        Globals.sealFlattenerFingersCount := Globals.sealFlattenerFingersCount +1;
    SEAL_FLATTENER_STATES.Ready :
    SEAL_FLATTENER_STATES.Fault :
END_CASE

METHOD AutoMoveIn : BOOL
VAR_INPUT
END_VAR
_amMoveIn := TRUE;
END_METHOD

METHOD AutoMoveToBagHolding
VAR_INPUT
END_VAR
_amMoveInToBagHolding := TRUE;
END_METHOD

METHOD AutoMoveToHandLoad : BOOL
VAR_INPUT
END_VAR
_amMoveHandLoad := TRUE;
END_METHOD

PROPERTY Ready : BOOL
SET
_ready := Ready;
END_SET
GET
Ready := _ready;
END_GET
END_PROPERTY

PROPERTY Mode : DEVICE_MODES
SET
_mode := Mode;
END_SET
GET
Mode := _mode;
END_GET
END_PROPERTY

METHOD PRIVATE ClearCommands
VAR_INPUT
END_VAR
// Clear all commands from auto mode
_amMoveOut := FALSE;
_amMoveClearance := FALSE;
_amMoveInToBagHolding := FALSE;
_amMoveIn := FALSE;
_amMoveHandLoad := FALSE;
END_METHOD

METHOD AutoMoveToClearance
VAR_INPUT
END_VAR
_amMoveClearance := TRUE;
END_METHOD

METHOD AutoMoveOut
VAR_INPUT
END_VAR
_amMoveOut := TRUE;
END_METHOD

END_FUNCTION_BLOCK

// FBs/Components/MotorizedSealFlattenersFB
FUNCTION_BLOCK MotorizedSealFlattenersFB EXTENDS BaseComponentFB IMPLEMENTS IComponentStatus
VAR_INPUT
    {warning 'TODO: Make a struct for some of these - too many inputs'}
	sealFlattenersVerticalAxis : ICylinder();
    clearanceOffset : REAL := 0.75;        // Clearance Offset in inches
    inSetpoint : REAL := 1.25;            // In setpoint in inches
    outSetpoint : REAL := 17.7;            // Out (sealing) setpoint in inches
    bagHoldingSetpoint : REAL := 17;    // Bag holding setpoint in inches            
    clearanceSpeed : INT := 3000;        // Speed to move in clearance move
    moveInSpeed : INT := 3000;            // Speed to move in in move
    moveOutSpeed : INT := 1000;            // Speed to move in out move
    moveBagHoldingSpeed : INT := 10000;    // Speed to move in bag holding move
    fingersUpSetpoint : REAL := 0;     // Fingers Up setpoint in inches
    fingersDownSetpoint : REAL := 1.1; // Fingers down setpoint in inches
    moveFingersSpeed : INT := 2000;        // Speed to move fingers
    horizontalAxisAccel : INT := 1000;    // Accel setpoint for horizontal axis
    horizontalAxisDecel : INT := 1000;    // Decel Setpoint for horizontal axis
    verticalAxisAccel : INT := 150;    // Accel setpoint for vertical axis
    verticalAxisDecel : INT := 150;    // Decel Setpoint for vertical axis
    testMovePB : BOOL;
    testMoveSP : REAL;
    stopPB : BOOL;
    startPB : BOOL;
    nextSeqPB : BOOL;
    delay : TON := (PT:= T#300MS);
	fingersDownDelay : Standard.TON := (PT := T#200MS);
	
	manualPosSetpoint : REAL;
	
END_VAR
VAR_IN_OUT
	jogIn : BOOL;
	jogOut : BOOL;
	raiseService : BOOL;
	lowerService : BOOL;
	moveToManualSetpoint : BOOL;
END_VAR
VAR_OUTPUT
    state : SEAL_FLATTENER_STATES;
END_VAR
VAR
    //pressureBarMotor : FB_FestoMotor();
    //sealFlattenersVerticalAxisMotor : FB_AppliedMotionStepServoRTU();
	jogInONS: FB_ONS;
	jogOutONS: FB_ONS;
	jogSpeed : INT := 100;
    sealFlattenersHorizontalAxisMotor : FB_AppliedMotionStepServoEIPBaseQX();
	defaultCurrentMSF : DINT := 150;
	outCurrentMSF : DINT := 150;
	bagHoldingCurrentMSF : DINT := 85;
    enableMotorizedSealFlattenersONS : R_TRIG();    
    _amMoveOut : BOOL;                // Auto mode move out command
	_amMoveIn : BOOL;
    _amMoveClearance : BOOL;            // Auto mode move Clearance command
    _amMoveInToBagHolding : BOOL;    // Auto mode move in then bag holding command
END_VAR

//    Function Block:  MotorizedSealFlattenersFB
//    Description: State machine and motor management for motorized seal flateners
//    Currently, this code requires one to use the Oriental drive with pre-programmed 
//    sequence for the horizontal axis
//    Created by: Ben Hess
//    Created Date: Friday, April 6, 2018
SUPER^();
// Setup and execute 2 motor axis'

// Temporary delay between states for testing
fingersDownDelay();
delay();
jogInONS(CLK := jogIn);
jogOutONS(CLK := jogOut);
IF autoModeSelected THEN
    delay.PT := T#300MS;
ELSE
    delay.PT := T#750MS;
END_IF

outSetpoint := HMIData.bagWidth + 0.2;
bagHoldingSetpoint := HMIData.bagWidth;

// Setup the vertical axis motor
sealFlattenersVerticalAxis.Execute();

// Setup the horizontal axis motor 
(*
sealFlattenersHorizontalAxisMotor(modbusInBuffer := OrientalMotorModbusRead,
                stepsPerInchSetpoint := 125,
                reversePolarity := FALSE,
                operatingCurrentDefault := 500,
                modbusCommandOutBuffer := OrientalMotorCommandWrites,
                modbusParametersOutBuffer := OrientalMotorParameterWrites,
                triggerCommandWrite => OrientalMotorTriggerCommandWrite,
                triggerParameterWrite => OrientalMotorTriggerParameterWrite);                
sealFlattenersHorizontalAxisMotor.Execute();
*)

sealFlattenersHorizontalAxisMotor(ptrEIPInputs := ADR(sealFlattenerHorizontalMotorInputs),
                ptrEIPOutputs := ADR(sealFlattenerHorizontalMotorOutputs),
                stepsPerInchSetpoint := Globals.STEPS_PER_INCH_SEAL_FLATTENER_HORIZONTAL_AXIS_MOTOR,
                faultHandler := PRG_Bagger.faultHandler,
				reversePolarity := TRUE, 
				defaultCurrentSetpoint := defaultCurrentMSF, 
				commFail := MSFMotor.eState <> IoDrvEthernetIP.AdapterState.RUNNING,
				isHomable := TRUE);
				
sealFlattenersHorizontalAxisMotor.Execute();

//Report as ready if mode is auto and we're not faulted
_ready := (_mode = DEVICE_MODES.Auto) AND NOT (state = SEAL_FLATTENER_STATES.Fault);

enableMotorizedSealFlattenersONS(CLK := enable);
IF stopPB THEN
    sealFlattenersHorizontalAxisMotor.Stop();
    stopPB := FALSE;
END_IF

IF startPB AND semiAutoModeSelected THEN 
    //sealFlattenersHorizontalAxisMotor.StartOperation();
    startPB := FALSE;
END_IF

IF nextSeqPB THEN 
    //sealFlattenersHorizontalAxisMotor.NextSequence();
    nextSeqPB := FALSE;
END_IF

IF testMovePB THEN
    sealFlattenersHorizontalAxisMotor.MoveToPosition(position := (testMoveSP), acceleration := 100, deceleration := 100, velocity := 600);
    testMovePB := FALSE;
END_IF

IF enableONS.Q OR resetONS.Q THEN 
    state := SEAL_FLATTENER_STATES.Idle;
	sealFlattenersHorizontalAxisMotor.Reset();
	_reset := FALSE;
	ClearCommands();
END_IF

IF NOT enable THEN
    state := SEAL_FLATTENER_STATES.Fault;
END_IF

// State amchine for motorized seal flatteners
CASE state OF
    

    SEAL_FLATTENER_STATES.Idle :                                    //If enabled move to out
                                                                    IF enable AND semiAutoModeSelected OR (autoModeSelected AND _amMoveOut) THEN
                                                                        state := SEAL_FLATTENER_STATES.MoveFlattenersOut;
                                                                        ClearCommands();
                                                                    END_IF
																	
																	IF enable AND autoModeSelected AND _amMoveIn OR _amMoveInToBagHolding THEN
																	//IF enable AND autoModeSelected AND _amMoveIn THEN
																		sealFlattenersVerticalAxis.Retract();
																		state := SEAL_FLATTENER_STATES.MoveFlattenersIn;
																		ClearCommands();
																	END_IF
																	
																	IF jogInONS.OSR THEN
																		sealFlattenersHorizontalAxisMotor.MoveDistance(distance := -18, 
																									acceleration := horizontalAxisAccel, 
																									deceleration := horizontalAxisDecel, 
																									velocity := jogSpeed);
																	ELSIF jogOutONS.OSR THEN
																		sealFlattenersHorizontalAxisMotor.MoveDistance(distance := 18, 
																									acceleration := horizontalAxisAccel, 
																									deceleration := horizontalAxisDecel, 
																									velocity := jogSpeed);
																	ELSIF jogInONS.OSF OR jogOutONS.OSF THEN
																		sealFlattenersHorizontalAxisMotor.Stop();
																	END_IF
																	
																	IF raiseService THEN
																		sealFlattenersVerticalAxis.Retract();  
																		raiseService := FALSE;
																	ELSIF lowerService THEN
																		sealFlattenersVerticalAxis.Extend();  
																		lowerService := FALSE;
																	END_IF
																	
																	IF moveToManualSetpoint THEN
																		sealFlattenersHorizontalAxisMotor.MoveToPosition(position := manualPosSetpoint, 
																									acceleration := horizontalAxisAccel, 
																									deceleration := horizontalAxisDecel, 
																									velocity := moveFingersSpeed);
																		moveToManualSetpoint := FALSE;
																	END_IF
																	
                                                                    
    SEAL_FLATTENER_STATES.MoveFlattenersOut :                        // Move flatteners to out position
                                                                
                                                                    //sealFlattenersHorizontalAxisMotor.StartOperation();
                                                                    sealFlattenersHorizontalAxisMotor.MoveToPositionTorque(position := outSetpoint, 
                                                                                                                        acceleration := horizontalAxisAccel,
                                                                                                                        deceleration := horizontalAxisDecel,
                                                                                                                        velocity := moveOutSpeed,
																														current := outCurrentMSF);                                                    
                                                                    state := SEAL_FLATTENER_STATES.MovingFlattenersOut;
                                                                    
                                                                    
    SEAL_FLATTENER_STATES.MovingFlattenersOut :                        // 
                                                                    delay.IN := TRUE;
                                                                    IF delay.Q THEN
																		IF sealFlattenersHorizontalAxisMotor.CommandAcknowledged AND sealFlattenersHorizontalAxisMotor.CurrentPosition >= (bagHoldingSetpoint - 1.5) THEN
																			state := SEAL_FLATTENER_STATES.MovedFlattenersOut;
                                                                        	delay.IN := FALSE; 
																		END_IF
                                                                    END_IF
                                                                    
    SEAL_FLATTENER_STATES.MovedFlattenersOut :                        // Move flatteners to clearance position state
                                                                    IF enable AND semiAutoModeSelected OR (autoModeSelected AND _amMoveClearance) THEN
                                                                        state := SEAL_FLATTENER_STATES.MoveFlattenersUpAndToClearance;
                                                                        ClearCommands();
                                                                    END_IF
    
    
    SEAL_FLATTENER_STATES.MoveFlattenersUpAndToClearance :                // Move flatteners to clearance position
                                                                    
                                                                    //sealFlattenersHorizontalAxisMotor.NextSequence();
                                                                    sealFlattenersHorizontalAxisMotor.MoveToPosition(position := (outSetpoint - clearanceOffset), 
                                                                                                                        acceleration := horizontalAxisAccel,
                                                                                                                        deceleration := horizontalAxisDecel,
                                                                                                                        velocity := moveOutSpeed);    
                                                                   	sealFlattenersVerticalAxis.Retract();                                                       
                                                                    state := SEAL_FLATTENER_STATES.MovingFlattenersUpAndToClearance;    
    
    
    
    SEAL_FLATTENER_STATES.MovingFlattenersUpAndToClearance :        delay.IN := TRUE;
                                                                    IF delay.Q THEN
																		IF sealFlattenersHorizontalAxisMotor.CommandAcknowledged AND sealFlattenersHorizontalAxisMotor.InPosition THEN
																			state := SEAL_FLATTENER_STATES.MovedFlattenersUpAndToClearance;    
                                                                        	delay.IN := FALSE;
																		END_IF
                                                                    END_IF
                                                                    
                                                                    
    SEAL_FLATTENER_STATES.MovedFlattenersUpAndToClearance :                // Move flatteners to up state
                                                                    IF enable AND semiAutoModeSelected OR (autoModeSelected AND (_amMoveInToBagHolding OR _amMoveIn)) THEN
                                                                        state := SEAL_FLATTENER_STATES.MoveFlattenersIn;
                                                                        //ClearCommands();
                                                                    END_IF
                                        
                                                                    
    SEAL_FLATTENER_STATES.MoveFlattenersIn :                        // Move flatteners up and in
                                                                    //sealFlattenersHorizontalAxisMotor.NextSequence();    
                                                                    sealFlattenersHorizontalAxisMotor.MoveToPosition(position := inSetpoint, 
                                                                                                                        acceleration := horizontalAxisAccel,
                                                                                                                        deceleration := horizontalAxisDecel,
                                                                                                                        velocity := moveInSpeed);                                                    
                                                                    state := SEAL_FLATTENER_STATES.MovingFlattenersIn;
                                                                    
                                                                    
    SEAL_FLATTENER_STATES.MovingFlattenersIn :                        // If we did that command well move on 
                                                                        delay.IN := TRUE;
                                                                        IF delay.Q THEN
																			IF sealFlattenersHorizontalAxisMotor.CommandAcknowledged AND sealFlattenersHorizontalAxisMotor.InPosition THEN
																				state := SEAL_FLATTENER_STATES.MovedFlattenersIn;
                                                                           		delay.IN := FALSE;    
																			END_IF
                                                                        END_IF 
                                                                    
    SEAL_FLATTENER_STATES.MovedFlattenersIn :                        // Now that we're up and in move to down and 4 corners/bag holding
                                                                    IF enable AND semiAutoModeSelected OR (autoModeSelected AND _amMoveInToBagHolding) THEN
                                                                        state := SEAL_FLATTENER_STATES.MoveFlattenersDown;
                                                                        ClearCommands();
                                                                    END_IF    
    
    SEAL_FLATTENER_STATES.MoveFlattenersDown :            // Do moves for down and bag holding
                                                                        
                                                                        sealFlattenersVerticalAxis.Extend();
                                                                                                                                                                                
                                                                        state := SEAL_FLATTENER_STATES.MovingFlattenersDown;
                                                                        
    SEAL_FLATTENER_STATES.MovingFlattenersDown :            
                                                                        //IF sealFlattenersVerticalAxis.CommandAcknowledged AND sealFlattenersVerticalAxis.InPosition THEN
                                                                       	fingersDownDelay.IN := TRUE;
																	  	IF fingersDownDelay.Q THEN
																			state := SEAL_FLATTENER_STATES.MovedFlattenersDown;
																			fingersDownDelay.IN := FALSE;
																		END_IF 
																		
                                                                        //END_IF 
                                                                        
    SEAL_FLATTENER_STATES.MovedFlattenersDown :            state := SEAL_FLATTENER_STATES.MoveFlattenersToBagHolding;
                                                                    
                                                                    
    SEAL_FLATTENER_STATES.MoveFlattenersToBagHolding :            // Do moves for down and bag holding
                                                                        //sealFlattenersHorizontalAxisMotor.NextSequence();    
                                                                        sealFlattenersHorizontalAxisMotor.MoveToPositionTorque(position := bagHoldingSetpoint, 
                                                                                                                        acceleration := horizontalAxisAccel,
                                                                                                                        deceleration := horizontalAxisDecel,
                                                                                                                        velocity := moveBagHoldingSpeed,
																														current := bagHoldingCurrentMSF);                                                
                                                                        state := SEAL_FLATTENER_STATES.MovingFlattenersToBagHolding;
                                                                        
    SEAL_FLATTENER_STATES.MovingFlattenersToBagHolding :            delay.IN := TRUE;
                                                                        IF delay.Q THEN
																			IF sealFlattenersHorizontalAxisMotor.CommandAcknowledged THEN
																				state := SEAL_FLATTENER_STATES.MovedFlattenersToBagHolding;
                                                                            	delay.IN := FALSE; 
																			END_IF   
                                                                        END_IF 
                                                                        
    SEAL_FLATTENER_STATES.MovedFlattenersToBagHolding :            state := SEAL_FLATTENER_STATES.Idle;
																		HMIData.motorizedSealFlattenerCycles.Increment();
                                                                        Globals.motorizedSealFlattenersCount := Globals.motorizedSealFlattenersCount +1;
                                                                        Globals.sealFlattenerFingersCount := Globals.sealFlattenerFingersCount +1;
    SEAL_FLATTENER_STATES.Ready :
    SEAL_FLATTENER_STATES.Fault :
END_CASE

METHOD PRIVATE ClearCommands
VAR_INPUT
END_VAR
// Clear all commands from auto mode
_amMoveOut := FALSE;
_amMoveClearance := FALSE;
_amMoveInToBagHolding := FALSE;
_amMoveIn := FALSE;
END_METHOD

METHOD AutoMoveOut
VAR_INPUT
END_VAR
_amMoveOut := TRUE;
END_METHOD

PROPERTY Mode : DEVICE_MODES
SET
_mode := Mode;
END_SET
GET
Mode := _mode;
END_GET
END_PROPERTY

PROPERTY Ready : BOOL
GET
Ready := _ready;
END_GET
SET
_ready := Ready;
END_SET
END_PROPERTY

METHOD AutoMoveToClearance
VAR_INPUT
END_VAR
_amMoveClearance := TRUE;
END_METHOD

METHOD AutoMoveToBagHolding
VAR_INPUT
END_VAR
_amMoveInToBagHolding := TRUE;
END_METHOD

METHOD AutoMoveIn : BOOL
VAR_INPUT
END_VAR
_amMoveIn := TRUE;
END_METHOD

END_FUNCTION_BLOCK

// FBs/Cylinders/ICylinder
INTERFACE ICylinder

METHOD Extend
VAR_INPUT
END_VAR
END_METHOD

METHOD Execute
VAR_INPUT
END_VAR
END_METHOD

METHOD Retract
VAR_INPUT
END_VAR
END_METHOD

END_INTERFACE

// FBs/Motors/Festo/FB_FestoMotor
FUNCTION_BLOCK FB_FestoMotor IMPLEMENTS IPositionableMotor, IStoredProgramMotor
VAR_INPUT
    deviceType : FML.E_FML_DEVICE_TYPE;                            //Must define drive type
    isFPCActive : BOOL;    
    ptrReadFHPPRegister : POINTER TO WORD;
    ptrReadFPCRegister : POINTER TO WORD;
    ptrWriteFHPPRegister : POINTER TO WORD;
    ptrWriteFPCRegister : POINTER TO WORD;                                        //Toggle if FPC(Festo Parameter Chanel) is active or not
END_VAR
VAR_IN_OUT
    //modbusReadRegisters :  ARRAY[0..7] OF WORD;        //Inputs from drive
    //modbusWriteRegisters : ARRAY[0..7] OF WORD;    //Outputs to write to drive

END_VAR
VAR_OUTPUT
END_VAR
VAR
    //Required datatypes for the Festo motor blocks
    FHPP_IN     :ARRAY[0..7] OF BYTE;
    FHPP_OUT     :ARRAY[0..7] OF BYTE;
    FPC_IN         :ARRAY[0..7] OF BYTE;
    FPC_OUT     :ARRAY[0..7] OF BYTE;
    ReadAxis            :FML.FML_Read;
    DATA_REF_Axis         :FML.DT_FML_REF;
    CRTL_Axis            :FML.FHPP_CTRL;
    PNU_Axis            :FML.FPC_PNU;
    MULTI_Axis            :FML.FPC_MULTI;    
    DIRMP_Axis            :FML.FPC_DIRMP;
    DIAG_Axis            :FML.FPC_DIAG;
    DIAG_BUFF_Axis        :FML.FPC_DIAG_BUFFER;
    DATA_OBJECT_Axis    :FML.FPC_DATA_OBJECT;
    FILE_Axis            :FML.FPC_FILE;
    FILE_ARRAY_Axis        :FML.FPC_FILE_ARRAY;
    WriteAxis            :FML.FML_Write;

    //Regular variables
    ptrModbusMemory : POINTER TO ARRAY[0..7] OF BYTE; 
    commandSuccessful : BOOL;    //Modbus Command was successful
    homeRequiredIndication : BOOL; //Home required indication
    homingActive : BOOL;            //Homing active
    removeStartCommandTimer : Standard.TON := (PT := T#100MS);
    startAckONS : Standard.R_TRIG;
    _sendStart : BOOL;
END_VAR
VAR_STAT    
    //Make these static to share amongst all instances of the Festo motors
    ARY_DATA_FILE        :ARRAY[0..25000] OF BYTE;
    MultiParam             :ARRAY [0..7] OF DT_FML_PRM_DESCRIPTION :=[
                                            (PNU:=404, SUBINDEX:=1, ACCESS:=0, VALUE:=0, LENGTH:=0),
                                            (PNU:=404, SUBINDEX:=1, ACCESS:=1, VALUE:=100, LENGTH:=4),
                                            (PNU:=404, SUBINDEX:=1, ACCESS:=0, VALUE:=0, LENGTH:=0),
                                            (PNU:=404, SUBINDEX:=2, ACCESS:=0, VALUE:=0, LENGTH:=0),
                                            (PNU:=404, SUBINDEX:=2, ACCESS:=1, VALUE:=200, LENGTH:=4),
                                            (PNU:=404, SUBINDEX:=2, ACCESS:=0, VALUE:=0, LENGTH:=0),
                                            (PNU:=404, SUBINDEX:=1, ACCESS:=1, VALUE:=111, LENGTH:=4),
                                            (PNU:=404, SUBINDEX:=1, ACCESS:=0, VALUE:=0, LENGTH:=0)];
                                            
END_VAR

METHOD ExecuteStoredProgram
VAR_INPUT
    (*Program number to execute*)
    programNumber    : INT;
END_VAR
InitDrive();
IF InPosition AND CRTL_Axis.ActualRecordNo = programNumber THEN
    commandSuccessful := TRUE;
ELSE
    CRTL_Axis.RecordNo := programNumber;
    _sendStart := TRUE;
END_IF
END_METHOD

PROPERTY Homing : BOOL
GET
Homing := homingActive;
END_GET
END_PROPERTY

PROPERTY HomeRequired : BOOL
GET
HomeRequired := homeRequiredIndication;
END_GET
SET
homeRequiredIndication := HomeRequired;
END_SET
END_PROPERTY

{attribute 'monitoring' := 'variable'}
PROPERTY CurrentPosition : REAL
GET
{warning: 'TODO: Find out actual conversion factor'}    
CurrentPosition := (DINT_TO_REAL(CRTL_Axis.ActualPosition)/100);
END_GET
END_PROPERTY

METHOD Execute
VAR_INPUT
END_VAR


//Check to make sure we have a valid reference.  Disable complier warning since we're doing the check
//{warning disable C0371}
(*
IF NOT __ISVALIDREF(ptrReadFHPPRegister) 
    OR NOT __ISVALIDREF(ptrReadFPCRegister) 
    OR NOT __ISVALIDREF(ptrWriteFHPPRegister)
    OR NOT __ISVALIDREF(ptrWriteFPCRegister)
THEN
     RETURN;
END_IF
*)



//Convert array of bytes to array of words. Playin' with pointers!
ptrModbusMemory := ptrReadFHPPRegister;
FHPP_IN := ptrModbusMemory^; 
ptrModbusMemory := ptrReadFPCRegister;
FPC_IN := ptrModbusMemory^;
ptrModbusMemory := ptrWriteFHPPRegister;
ptrModbusMemory^ := FHPP_OUT; 
ptrModbusMemory := ptrWriteFPCRegister;
ptrModbusMemory^ := FPC_OUT;

// Function block calls for axis
ReadAxis(
    FML_REF            := DATA_REF_Axis,
    Modbus            := FALSE,
    HighByteFirst    := TRUE,
    DeviceType        := deviceType,
    FPC_active        := isFPCActive,
    
    FHPP_Source        := FHPP_IN,
    FPC_Source        := FPC_IN);    
CRTL_Axis(
    FML_REF            := DATA_REF_Axis);    
PNU_Axis(
    FML_REF            := DATA_REF_Axis);
MULTI_Axis(
    FML_REF            := DATA_REF_Axis,
    SizeOfParam        := SIZEOF(MultiParam),
    AdrOfParam        := ADR(MultiParam));
DIRMP_Axis(
    FML_REF            := DATA_REF_Axis);    
DIAG_Axis(
    FML_REF            := DATA_REF_Axis);
DIAG_BUFF_Axis(
    FML_REF            := DATA_REF_Axis);
DATA_OBJECT_Axis(
    FML_REF            := DATA_REF_Axis);
FILE_Axis(
    FML_REF            := DATA_REF_Axis);
FILE_ARRAY_Axis(
    FML_REF            := DATA_REF_Axis,
    SizeOfFileArray    := SIZEOF(ARY_DATA_FILE),
    AdrOfFileArray    := ADR(ARY_DATA_FILE));    
WriteAxis(
    FML_REF            := DATA_REF_Axis,
    FHPP_Target        => FHPP_OUT,
    FPC_Target        => FPC_OUT);
{warning 'TODO: Remove this hack to clear start command if error occurs'}
removeStartCommandTimer(IN := CRTL_Axis.StartTask OR CRTL_Axis.AckStart);
//removeStartCommandTimer(IN := CRTL_Axis.AckStart);
startAckONS(CLK := CRTL_Axis.AckStart);    
//IF removeStartCommandTimer.Q THEN
IF _sendStart AND NOT CRTL_Axis.AckStart THEN
    CRTL_Axis.StartTask := TRUE;
    _sendStart := FALSE;
END_IF

IF startAckONS.Q OR removeStartCommandTimer.Q THEN
    CRTL_Axis.StartTask := FALSE;
    commandSuccessful := TRUE;
END_IF
//Set Home required indication
homeRequiredIndication S= NOT CRTL_Axis.HomingValid;
//commandSuccessful S= CRTL_Axis.AckStart;
//{warning restore C0371}
END_METHOD

{attribute 'monitoring' := 'variable'}
PROPERTY CommandAcknowledged : BOOL
GET
CommandAcknowledged := commandSuccessful;
END_GET
END_PROPERTY

METHOD Stop
commandSuccessful := FALSE;
CRTL_Axis.EnableDrive := TRUE;
CRTL_Axis.Halt := TRUE;
CRTL_Axis.Stop := FALSE;
END_METHOD

{attribute 'monitoring' := 'variable'}
PROPERTY ActiveStoredProgramNumber : INT
GET
ActiveStoredProgramNumber := CRTL_Axis.ActualRecordNo;
END_GET
END_PROPERTY

METHOD PRIVATE InitDrive
VAR_INPUT
END_VAR
//Initialize the drive to prepare for a move
CRTL_Axis.EnableDrive := TRUE;
CRTL_Axis.Halt := TRUE;
CRTL_Axis.Stop := TRUE;    
//CRTL_Axis.StartTask := FALSE;
commandSuccessful := FALSE;
END_METHOD

PROPERTY Moving : BOOL
GET
Moving := CRTL_Axis.DriveIsMoving;
END_GET
END_PROPERTY

{warning 'add method implementation '}
METHOD MoveDistance
VAR_INPUT
    (*Distance to move in inches*)
    distance    : REAL;
    (*Acceleration in RPM/sec*)
    acceleration    : INT;
    (*Deceleration in RPM/sec*)
    deceleration    : INT;
    (*Velocity in .25RPM*)
    velocity    : INT;
END_VAR
END_METHOD

{attribute 'monitoring' := 'variable'}
PROPERTY InPosition : BOOL
GET
InPosition := CRTL_Axis.MC;
END_GET
END_PROPERTY

{warning 'add method implementation '}
METHOD MoveToPosition
VAR_INPUT
    (*Position to move to in inches*)
    position    : REAL;
    (*Acceleration in RPM/sec*)
    acceleration    : INT;
    (*Deceleration in RPM/sec*)
    deceleration    : INT;
    (*Velocity in .25RPM*)
    velocity    : INT;
END_VAR
END_METHOD

METHOD HomeNow
CRTL_Axis.StartHoming := TRUE;
END_METHOD

END_FUNCTION_BLOCK

// FBs/Motors/IPositionableMotor
INTERFACE IPositionableMotor

PROPERTY Homing : BOOL
GET
END_GET
END_PROPERTY

PROPERTY Moving : BOOL        //Motor is Moving
GET
END_GET
END_PROPERTY

PROPERTY InPosition : BOOL        //Motor is in position
GET
END_GET
END_PROPERTY

PROPERTY CurrentPosition : REAL        //Current motor position in Inches
GET
END_GET
END_PROPERTY

METHOD Stop
VAR_INPUT
END_VAR
END_METHOD

PROPERTY CommandAcknowledged : BOOL        //Command acked from drive
GET
END_GET
END_PROPERTY

METHOD HomeNow
VAR_INPUT
END_VAR
END_METHOD

METHOD MoveToPosition
VAR_INPUT
    position : REAL;        //Position to move to in inches
    acceleration : INT;        //Acceleration in RPM/sec
    deceleration : INT;        //Deceleration in RPM/sec
    velocity : INT;            //Velocity in .25RPM
END_VAR
END_METHOD

PROPERTY HomeRequired : BOOL
GET
END_GET
SET
END_SET
END_PROPERTY

METHOD MoveDistance
VAR_INPUT
    distance : REAL;        //Distance to move in inches
    acceleration : INT;        //Acceleration in RPM/sec
    deceleration : INT;        //Deceleration in RPM/sec
    velocity : INT;            //Velocity in .25RPM
END_VAR
END_METHOD

END_INTERFACE

// FBs/Motors/IStoredProgramMotor
INTERFACE IStoredProgramMotor

PROPERTY ActiveStoredProgramNumber : INT
GET
END_GET
END_PROPERTY

METHOD ExecuteStoredProgram
VAR_INPUT
    programNumber : INT;        //Program number to execute
END_VAR
END_METHOD

END_INTERFACE

// FBs/Fault/FB_ONS
FUNCTION_BLOCK FB_ONS
VAR_INPUT
	CLK : BOOL;
END_VAR
VAR_OUTPUT
	OSR : BOOL;
	OSF : BOOL;
END_VAR
VAR
	CLK_OSR : R_TRIG;
	CLK_OSF : F_TRIG;
END_VAR

CLK_OSR(CLK := CLK, Q=> OSR);
CLK_OSF(CLK := CLK, Q=> OSF);

END_FUNCTION_BLOCK

// FBs/Motors/Applied Motion/FB_AppliedMotionStepServoEIPBaseQX
FUNCTION_BLOCK FB_AppliedMotionStepServoEIPBaseQX IMPLEMENTS IPositionableMotor, IStoredProgramMotor
VAR_INPUT
    ptrEIPInputs : POINTER TO ARRAY[0..13] OF  DINT;
    ptrEIPOutputs : POINTER TO ARRAY[0..15] OF DINT;
    faultHandler : REFERENCE TO FB_FaultHandler;
	commFail : BOOL;
    stepsPerInchSetpoint : INT;             //Steps per inch setpoint
    reversePolarity : BOOL;                 //0 = Normal, 1 = reversed polarity for display
    jogAccelSetpoint : INT;        //Point-to-Point Acceleration (AC) Setpoint
    jogDecelSetpoint : INT;        //Point-to-Point Deceleration (DE) Setpoint
    jogVelocitySetpoint : INT;                //Velocity (VE) Setpoint
    pointToPointAccelSetpoint : INT;        //Point-to-Point Acceleration (AC) Setpoint
    pointToPointDecelSetpoint : INT;        //Point-to-Point Deceleration (DE) Setpoint
    velocitySetpoint : INT;                //Velocity (VE) Setpoint
	defaultCurrentSetpoint : DINT;
	sclCommand : DINT;						// SCL Command from 
	parameter1 : DINT;						// Data/SCL parameter 1
	parameter2 : DINT;						// Data/SCL parameter 2
    distanceSetpointInches : REAL;        //Distance setpoint in inches Setpoint
    moveDistanceManualPB : BOOL;            //Move distance pushbutton
    movePositionManualPB : BOOL;            //Move position pushbutton
	isHomable : BOOL;
END_VAR
VAR_IN_OUT
    //slave : IoDrvModbusTCP.ModbusTCPSlave;                    //Slave ModbusTCP Object
END_VAR
VAR
    absolutePositionSteps : DINT; //Immediate Absolute Position in steps
    distanceToMoveInSteps : DINT;        //Distance Setpoint to Drive
    stepServoStatusRaw : INT; //Raw step servo status over modbus
	stepServoAlarmCodeRaw : INT; // Ras Step Servo alarm code word
	currentLimit : DINT;
    commands : FB_StepServoCommands();
    commandSuccessful : BOOL;    //Modbus Command was successful
    commandSuccessfulONS : R_TRIG;    //Modbus Command was successful
    commandSentONS : R_TRIG;    //Modbus Command was successful
    homeRequiredIndication : BOOL; //Home required indication.
    driveInputs : ARRAY[0..13] OF DINT;        // Inputs from drive over EIP
    driveOutputs : ARRAY[0..15] OF DINT;    // Outputs to drive over EIP
    interfaceToPass : IFault;
    faultListRegisterSuccess : BOOL;        // Registering in fault list successful
    _faulted : BOOL;                    // Motor Faulted
	_reset : BOOL;			//Reset Motor
	_homeNow : BOOL;
	homingOSF : F_TRIG;
	
	IECReferenceGood : BOOL;
END_VAR
VAR_OUTPUT
    absolutePositonInches : REAL; //Immediate Absolute Positon in inches
    velocity : INT;    //Velocity (VE) Input from Drive
    status : StepServoStatusFB; //Status of servo
	alarms : FB_StepServoAlarms; // Alarms from Drive
    QSegmentRunning : INT; //Current Q program running from Drive
	faults : StepServoFaultsType;
END_VAR


IF NOT faultListRegisterSuccess THEN
    faultListRegisterSuccess := RegisterWithFaultHandler();
END_IF

METHOD Execute
VAR_INPUT
END_VAR
//    Function Block: AppliedMotionStepServo
//    Description: This block provides an abstraction for a Ethernet I/P Applied Motion Step Servo
//    Created by: Ben Hess
//    Created Date: May 11th, 2018

// Use pointers for EIP memory register locations
driveInputs := ptrEIPInputs^;

ptrEIPOutputs^ := driveOutputs;
alarms(alarmCode := stepServoAlarmCodeRaw, faults := faults);

IF currentLimit = 0 THEN 
	currentLimit := defaultCurrentSetpoint;
END_IF
//Map raw EIP Registers to parameters
absolutePositionSteps := driveInputs[6];
velocity := DINT_TO_INT(driveInputs[8]);
stepServoStatusRaw := DINT_TO_INT(driveInputs[0]);

driveOutputs[4] := velocitySetpoint;
driveOutputs[5] := pointToPointAccelSetpoint;
driveOutputs[6] := pointToPointDecelSetpoint;
driveOutputs[7] := distanceToMoveInSteps;
driveOutputs[8] := currentLimit;
driveOutputs[9] := sclCommand;
driveOutputs[10] := parameter1;
driveOutputs[11] := parameter2;
driveOutputs[12] := currentLimit;
driveOutputs[13] := currentLimit + 1;
driveOutputs[0] := commands.commandWord;
// Step servo command bits handler
commands();
//Convert Distance setpoint to steps.  Reverse polarity for display purposes if needed. 

absolutePositonInches := (DINT_TO_REAL(absolutePositionSteps) / INT_TO_REAL(stepsPerInchSetpoint));

//Homing required from motor - for now just if there was an initialization seen.
homeRequiredIndication S= status.initializing OR Globals.firstScan OR _faulted OR driveInputs[11].0;

homingOSF(CLK := status.homing);
IF NOT driveInputs[11].0 THEN
	homeRequiredIndication := FALSE;
END_IF

commandSentONS(CLK := commands.commandSent);

IF commandSentONS.Q THEN
	commandSuccessful := TRUE;
END_IF

commandSuccessfulONS(CLK := commandSuccessful);
IF commandSuccessfulONS.Q THEN
	//parameter1 := 0;
	//velocitySetpoint := 0;
	//pointToPointAccelSetpoint := 0;
	//pointToPointDecelSetpoint := 0;
	//distanceToMoveInSteps := 0;
END_IF


IF _reset AND (status.driveFaulted OR status.alarmPresent) THEN
	commands.alarmReset := TRUE;
	_reset := FALSE;
END_IF

IF reversePolarity THEN
    absolutePositonInches := absolutePositonInches * -1; 
END_IF

//Get Servo Status and unpack
status(statusCode := StepServoStatusRaw);

//Bit-packing for LONG types over Modbus

_faulted := status.driveFaulted OR status.alarmPresent OR commFail;

//Manual moves for motor
IF moveDistanceManualPB THEN
    MoveDistance(distance := distanceSetpointInches, acceleration := pointToPointAccelSetpoint, deceleration := pointToPointDecelSetpoint, velocity := velocitySetpoint);
    moveDistanceManualPB := FALSE;
END_IF

IF movePositionManualPB THEN
    MoveToPosition(position := distanceSetpointInches, acceleration := pointToPointAccelSetpoint, deceleration := pointToPointDecelSetpoint, velocity := velocitySetpoint);
    movePositionManualPB := FALSE;
END_IF


faults.commFail.faultTrigger := commFail AND Globals.machinePowerOK;
faults.notHomed.faultTrigger := homeRequiredIndication AND isHomable;
END_METHOD

{attribute 'monitoring' := 'variable'}
PROPERTY CommandAcknowledged : BOOL
GET
CommandAcknowledged := commandSuccessful;
END_GET
END_PROPERTY

METHOD HomeNow
commandSuccessful := FALSE;
parameter1 := 1;
pointToPointAccelSetpoint := 1000;
pointToPointDecelSetpoint := 1000;
velocitySetpoint := 2500;
distanceToMoveInSteps := 0;
commands.sendQAndExecute := TRUE;

//homeRequiredIndication := FALSE;
END_METHOD

{attribute 'monitoring' := 'variable'}
PROPERTY HomeRequired : BOOL
SET
homeRequiredIndication := HomeRequired;
END_SET
GET
HomeRequired := homeRequiredIndication;
END_GET
END_PROPERTY

{attribute 'monitoring' := 'variable'}
PROPERTY Moving : BOOL
GET
Moving := status.moving;
END_GET
END_PROPERTY

{attribute 'monitoring' := 'variable'}
PROPERTY ActiveStoredProgramNumber : INT
GET
ActiveStoredProgramNumber := QSegmentRunning;
END_GET
END_PROPERTY

{attribute 'monitoring' := 'variable'}
PROPERTY InPosition : BOOL
GET
InPosition := status.inPosition;
END_GET
END_PROPERTY

METHOD MoveDistanceTorque
VAR_INPUT
	(*Distance to move in inches*)
    distance    : REAL;
    (*Acceleration in RPM/sec*)
    acceleration    : INT;
    (*Deceleration in RPM/sec*)
    deceleration    : INT;
    (*Velocity in .25RPM*)
    velocity    : INT;
	(*Current in .01A*)
	current : DINT;
END_VAR
//This method preps the data to send to the drive and triggers the send.
//Set distance and unpack to prep data to send to motor

commandSuccessful := FALSE;

distanceToMoveInSteps := REAL_TO_DINT((distance) * stepsPerInchSetpoint);
IF reversePolarity THEN
    distanceToMoveInSteps := distanceToMoveInSteps * -1;
END_IF

pointToPointAccelSetpoint := acceleration;
pointToPointDecelSetpoint := deceleration;
velocitySetpoint := velocity;
currentLimit := current;

parameter1 := 2;
commands.SendQAndExecute := TRUE;
END_METHOD

(* This will be called if the machine is faulted*)
METHOD MachineFaulted
END_METHOD

{attribute 'monitoring' := 'variable'}
PROPERTY Faulted : BOOL
GET
Faulted := _faulted;
END_GET
SET
END_SET
END_PROPERTY

METHOD MoveToPosition
VAR_INPUT
    (*Position to move to in inches*)
    position    : REAL;
    (*Acceleration in RPM/sec*)
    acceleration    : INT;
    (*Deceleration in RPM/sec*)
    deceleration    : INT;
    (*Velocity in .25RPM*)
    velocity    : INT;
END_VAR
commandSuccessful := FALSE;

distanceToMoveInSteps := REAL_TO_DINT((position) * stepsPerInchSetpoint);
IF reversePolarity THEN
    distanceToMoveInSteps := distanceToMoveInSteps * -1;    
END_IF

pointToPointAccelSetpoint := acceleration;
pointToPointDecelSetpoint := deceleration;
velocitySetpoint := velocity;
currentLimit := defaultCurrentSetpoint;

commands.feedToPosition := TRUE;
END_METHOD

METHOD MoveToPositionTorque
VAR_INPUT
	(*Position to move to in inches*)
    position    : REAL;
    (*Acceleration in RPM/sec*)
    acceleration    : INT;
    (*Deceleration in RPM/sec*)
    deceleration    : INT;
    (*Velocity in .25RPM*)
    velocity    : INT;
	(*Current in .01A*)
	current : DINT;
END_VAR
commandSuccessful := FALSE;

distanceToMoveInSteps := REAL_TO_DINT((position) * stepsPerInchSetpoint);
IF reversePolarity THEN
    distanceToMoveInSteps := distanceToMoveInSteps * -1;    
END_IF

pointToPointAccelSetpoint := acceleration;
pointToPointDecelSetpoint := deceleration;
velocitySetpoint := velocity;
currentLimit := current;

commands.feedToPosition := TRUE;
THIS^.Execute();
END_METHOD

//{warning 'add method implementation '}
METHOD Stop
commandSuccessful := FALSE;
commands.StopNormal := TRUE;
END_METHOD

METHOD MoveDistance
VAR_INPUT
    (*Distance to move in inches*)
    distance    : REAL;
    (*Acceleration in RPM/sec*)
    acceleration    : INT;
    (*Deceleration in RPM/sec*)
    deceleration    : INT;
    (*Velocity in .25RPM*)
    velocity    : INT;
END_VAR
//This method preps the data to send to the drive and triggers the send.
//Set distance and unpack to prep data to send to motor

commandSuccessful := FALSE;

distanceToMoveInSteps := REAL_TO_DINT((distance) * stepsPerInchSetpoint);
IF reversePolarity THEN
    distanceToMoveInSteps := distanceToMoveInSteps * -1;
END_IF

